(* IEC 61131-3 sources: LStream-JSON-XML/src/LStream (part 2) *)

(* ---- LStream_XmlDeserializer.st ---- *)
//region BLOCK INFO HEADER
    //===============================================================================
    // SIEMENS AG / (c)Copyright 2024
    //-------------------------------------------------------------------------------
    // Title:            LStream_XmlDeserializer
    // Comment/Function: parses a XML string provided in the Raw parameter
    //                   and rebuilds the contained tree structure
    // Library/Family:   LStream
    // Author:           DI FA S SUP E&C
    // Tested with:      S7-1500 V3.1
    // Engineering:      Simatic AX
    // Restrictions:     --
    // Requirements:     LStream_FindStringInByteArrayAdv(FC), LStream_typeElement(UDT)
    //-------------------------------------------------------------------------------
    // Change log table:
    // Version  | Date       | Expert in charge | Changes applied
    //----------|------------|------------------|------------------------------------
    // 01.00.00 | 2021-03-10 | DI FA S SUP E&C  | First released version
    // 01.06.00 | 2023-04-10 | DI FA S SUP E&C  | Rework and refactoring of entire library
    // 02.00.00 | 2024-11-11 | DI FA S SUP E&C  | Migrate library to Simatic AX
    //===============================================================================

//end_region
USING System.Timer;
USING System.Strings;
USING Simatic.Ax.LStream.Utilities;
USING Simatic.Ax.LStream.Models;
NAMESPACE Simatic.Ax.LStream
    FUNCTION_BLOCK LStream_XmlDeserializer
        VAR_INPUT
            /// Rising edge starts action once
            execute : BOOL;
            /// TRUE: Searches raw data for the value of the provided tree keys
            search  : BOOL;
        END_VAR
        VAR_OUTPUT
            /// TRUE: Commanded functionality has been completed successfully
            done : BOOL;
            /// TRUE: FB is not finished and new output values can be expected
            busy : BOOL;
            /// TRUE: An error occurred during the execution of the FB
            error : BOOL;
            /// 16#0000 - 16#7FFF: Status of the FB, 16#8000 - 16#FFFF: Error identification
            status : WORD := STATUS_NO_CALL;
            /// Current parse position in the raw XML data
            pointer : DINT;
            /// Count of parsed XML elements
            resultCount : DINT;
        END_VAR
        VAR_IN_OUT
            /// Tree parsed information is written to, if search option active, keys must be provided
            tree : ARRAY [*] of LStream_typeElement;
            /// Byte array of raw xml data
            raw : ARRAY[*] of BYTE;
        END_VAR
        VAR PUBLIC
            TimeoutTimer : System.Timer.OnDelay;
        END_VAR
        VAR
            /// Old value of 'execute' input for edge detection
            statOldExecute : BOOL;
            /// Static value of xml depth
            statDepth : SINT := SINT#-1;
            /// Static value of error
            statError : BOOL;
            /// Static value of busy
            statBusy : BOOL;
            /// Static value of status
            statStatus : WORD := STATUS_NO_CALL;
            /// Static value of fb state
            statFBState : USINT := FB_STATE_NO_PROCESSING;
            /// Static value of done
            statDone : BOOL;
            /// Static value of result count
            statResultCount : UINT;
            /// Static value of raw index
            statRawIndex : INT;
            /// Static value of tree index
            statTreeIndex : UINT;
            /// Static count of tree fields
            statCountOfTree : INT;
            /// Static count of raw fields
            statCountOfRaw : INT;
            /// TRUE: key is open, internal flag
            statIsKeyOpen : BOOL;
            /// TRUE: value is open, internal flag
            statIsValueOpen : BOOL;
            /// Determines the amount of open elements; if larger than 0 then at least one element is still open at the current parse position
            statElementOpen : UINT;
            /// TRUE: element is open, internal flag
            statIsElementOpen : BOOL;
            /// Current  information length key or value
            statInfoLen : UINT;
            /// Start index of current info in raw key or value
            statInfoStartIndex : INT;
            /// TRUE: Current key has already been written to the tree
            statKeyWritten: BOOL;
            /// Static key string
            statKey : STRING;
            /// Static value string
            statValue : STRING;
            /// TRUE: Only keys provided in tree will be parsed
            statSearch : BOOL;
            /// TRUE: Key exists in raw data
            statKeyFound : BOOL;
            /// Count of provided keys that weren't found
            statKeyNotFoundCount : UINT;
            /// Static search index
            statSearchIndex : DINT;
            /// Backtrack array for getting the last elements open
            statOpenElements : ARRAY[0.. MAX_CONCURRENT_OPEN_ELEMENTS] of UINT;
            /// Delimiter for attributes
            statAttrDelimiter : BYTE := BYTE#00;
        END_VAR
        VAR_TEMP
            /// Index of raw field
            tempRawIndex : INT;
            /// Temp of input execute
            tempExecute : BOOL;
            /// Provided key to which the value should be found
            tempKeyToFind : STRING;
            /// Temp value of search result
            tempSearchResult : DINT;
            /// Temp value of a byte for searching / looping
            tempChar : BYTE;
        END_VAR
        VAR CONSTANT
            /// FB state no processing, ideal state
            FB_STATE_NO_PROCESSING : USINT := USINT#0;
            /// FB state parse xml
            FB_STATE_PARSE : USINT := USINT#10;
            /// NO error - execution finished without errors
            STATUS_EXECUTION_FINISHED : WORD := WORD#16#0000;
            /// No job being currently processed
            STATUS_NO_CALL : WORD := WORD#16#7000;
            /// First call after incoming new job (rising edge 'execute')
            STATUS_FIRST_CALL : WORD := WORD#16#7001;
            /// Subsequent call during active processing without further details
            STATUS_SUBSEQUENT_CALL : WORD := WORD#16#7002;
            /// Error: provided array to too small
            ERR_TREE_ARRAY_TOO_SMALL : WORD := WORD#16#8201;
            /// Error: no raw data provided
            ERR_EMPTY_RAW_DATA : WORD := WORD#16#8401;
            /// Error: Encountered more closing tags than there are opening tags
            ERR_UNMATCHED_ELEMENT_CLOSE : WORD := WORD#16#8402;
            /// Error: Encountered an unexpected quotes character
            ERR_UNEXPECTED_QUOTES : WORD := WORD#16#8404;
            /// Error: Collection of all not further specified errors, e.g. unclosed elements before file end etc.
            ERR_MALFORMED : WORD := WORD#16#8406;
            /// Error: due to an undefined state in state machine
            ERR_UNDEFINED_STATE : WORD := WORD#16#8600;
            /// ASCII code for Unit Separator which is numerically the highest control character
            CONTROL_CHARACTERS_UPPER : WORD := WORD#16#1F;
            /// ASCII code for ? indicates xml header
            QUESTIONMARK : BYTE := BYTE#16#3F;
            /// ASCII code for ! indicates comment
            EXCLAMATION : BYTE := BYTE#16#21;
            /// ASCII code for " frames value
            DOUBLE_QUOTES : BYTE := BYTE#16#22;
            /// ASCII code for ' frames value
            QUOTES : BYTE := BYTE#16#27;
            /// ASCII code for < indicates a new key
            SMALLER : BYTE := BYTE#16#3C;
            /// ASCII code for '=' indicates key is finished follows by value
            EQUALS : BYTE := BYTE#16#3D;
            /// ASCII code for  > indicates key can be written
            GREATER : BYTE := BYTE#16#3E;
            /// ASCII code for SPACE indicates key is finished
            SPACE : BYTE := BYTE#16#20;
            /// ASCII code for / indicates closing
            SLASH : BYTE := BYTE#16#2F;
            /// ASCII code for carriage return
            CARRIAGE_RETURN : BYTE := BYTE#16#0D;
            /// ASCII code for line feed
            LINE_FEED : BYTE := BYTE#16#0A;
            /// ASCII code for TAB
            TAB : BYTE := BYTE#16#09;
            /// ASCII code for -
            MINUS : BYTE := BYTE#16#2D;
            /// Constant for zero value
            EMPTY : SINT := SINT#0;
            /// Numerical identifier for XML type element
            ELEMENT : SINT := SINT#0;
            /// Numerical identifier for XML type attribute
            ATTRIBUTE : SINT := SINT#1;
            /// Constant for first array dimension
            FIRST_DIM : USINT := USINT#1;
            /// Max duration of loop, will be continued in next cycle
            MAX_LOOP_TIME : TIME := T#3ms;
            /// Return value if Search in LStream_FindStringInByteCharArrayAdv was not successful
            INVALID_SEARCH : DINT := -1;
            /// String value in case key wasn't found
            KEY_NOT_FOUND : STRING := 'Key not found';
            /// String is default empty with string content named 'NULL'
            STRING_NULL : STRING := 'NULL';
            /// Maximal number of elements that can be open at any time
            MAX_CONCURRENT_OPEN_ELEMENTS : UINT := UINT#150;
            /// Empty string for resetting of fields
            STRING_EMPTY : STRING := '';

            /// ASCII code for ?
            QUESTIONMARK_INT : INT := 63;
            /// ASCII code for !
            EXCLAMATION_INT : INT := 33;
            /// ASCII code for "
            DOUBLE_QUOTES_INT : INT := 34;
            /// ASCII code for '
            QUOTES_INT : INT := 39;
            /// ASCII code for <
            SMALLER_INT : INT := 60;
            /// ASCII code for =
            EQUALS_INT : INT := 61;
            /// ASCII code for >
            GREATER_INT : INT := 62;
            /// ASCII code for SPACE
            SPACE_INT : INT := 32;
            /// ASCII code for /
            SLASH_INT : INT := 47;
            /// ASCII code for carriage return
            CARRIAGE_RETURN_INT : INT := 13;
            /// ASCII code for line feed
            LINE_FEED_INT : INT := 10;
            /// ASCII code for TAB
            TAB_INT : INT := 9;
            /// ASCII code for -
            MINUS_INT : INT := 45;
        END_VAR
        tempExecute := execute;

    //region TRIGGERING

        IF ((tempExecute = TRUE) AND (statOldExecute = FALSE) AND (statStatus = STATUS_NO_CALL)) THEN

            //First call; Initialize FB
            statDone := FALSE;
            statBusy := TRUE;
            statStatus := STATUS_FIRST_CALL;

            //Initialize functionality: reset of variables, diagnostics, etc.
            statSearch := search;
            statCountOfRaw := TO_INT(UPPER_BOUND(raw, FIRST_DIM));
            statCountOfTree := TO_INT(UPPER_BOUND(tree, FIRST_DIM));
            statTreeIndex := TO_UINT(LOWER_BOUND(tree, FIRST_DIM));
            statDepth := SINT#0;
            statRawIndex := 0;
            statIsKeyOpen := FALSE;
            statIsValueOpen := FALSE;
            statIsElementOpen := FALSE;
            statElementOpen := UINT#0;
            statKeyWritten := FALSE;
            statInfoLen := UINT#0;
            statInfoStartIndex := 0;
            statKey := '';
            statValue := '';
            statKeyFound := FALSE;
            statSearchIndex := 0;
            statKeyNotFoundCount := UINT#0;

            // State machine - start processing
            statFBState := FB_STATE_PARSE;

            IF (NOT (statCountOfRaw > EMPTY)) THEN
                statStatus := ERR_EMPTY_RAW_DATA;
            END_IF;

            FOR tempRawIndex := TO_INT(statTreeIndex) TO statCountOfTree DO

                tree[tempRawIndex].types := SINT#-1;
                tree[tempRawIndex].depth := SINT#-1;
                tree[tempRawIndex].key := STRING_EMPTY;
                tree[tempRawIndex].value := STRING_NULL;

            END_FOR;
        ELSIF (statStatus = STATUS_FIRST_CALL) THEN
            statStatus := STATUS_SUBSEQUENT_CALL;
        END_IF;

        // Edge detection 'execute' input
        statOldExecute := tempExecute;

    //endRegion TRIGGERING
        IF (statStatus = STATUS_NO_CALL) THEN // Nothing to do -> End here to reduce "system load"
            RETURN;
        END_IF;
    //region PROGRAM LOGIC

        CASE statFBState OF
            FB_STATE_NO_PROCESSING:
                // #region NO PROCESSING
                    // No processing active (Note: this state must always be present AND left empty)
                    ;
                // #endregion NO PROCESSING
            FB_STATE_PARSE:
                // #region PARSE XML

                    //reset and start watchdog here so that for loop runs for a maximum of 5 seconds
                    TimeoutTimer(signal := FALSE, duration := MAX_LOOP_TIME);

                    //start watchdog
                    TimeoutTimer(signal := TRUE, duration := MAX_LOOP_TIME);

                    tempRawIndex := statRawIndex;

                    WHILE tempRawIndex <= statCountOfRaw DO
                        //pre check if key exist in raw data, only if search option is active and key wasn't already found
                        IF (statSearch AND statKeyFound = FALSE) THEN
                            IF (TO_DINT(statTreeIndex) < statCountOfTree) THEN              //Convert to DINT to prevent possible overflows
                                tempSearchResult := LStream_FindStringInByteCharArrayAdv(searchFor := tree[statTreeIndex].key, startPosition := statSearchIndex, searchIn := raw);

                                IF tempSearchResult = INVALID_SEARCH THEN
                                    // Case key not found
                                    tree[statTreeIndex].value := KEY_NOT_FOUND;
                                    statTreeIndex := statTreeIndex + UINT#1;
                                    statKeyNotFoundCount := statKeyNotFoundCount + UINT#1;
                                ELSE
                                    // Case key found
                                    // move read pointer to last found index
                                    statSearchIndex := tempSearchResult;
                                    statKeyFound := TRUE;
                                END_IF;
                            END_IF;
                        END_IF;

                        statRawIndex := tempRawIndex;
                        // Switch case of current byte
                        CASE TO_INT(raw[tempRawIndex]) OF           //BYTE/ WORD Can not be selected as CASE selector
                            SMALLER_INT:
                                //region READ OPENING KEY SYMBOLS

                                    // There MUST be some characters after an open <
                                    // so if the array is too short the xml is malformed
                                    IF ((tempRawIndex + 1) > statCountOfRaw) THEN
                                        statStatus := ERR_MALFORMED;
                                        statDone := TRUE;
                                        EXIT;
                                    END_IF;
                                    IF statIsValueOpen
                                        AND statInfoLen > UINT#0
                                        AND tree[statOpenElements[statElementOpen]].value = STRING_NULL
                                        AND raw[statInfoStartIndex] <> SMALLER
                                    THEN
                                        //region WRITE VALUE
                                        IF statInfoLen < UINT#0 THEN
                                            statValue := STRING_EMPTY;
                                        ELSE
                                            CharsToString(chars := raw,
                                                        startPosition := statInfoStartIndex,
                                                        length:= statInfoLen,
                                                        result => statValue);
                                        END_IF;

                                        tree[statOpenElements[statElementOpen]].value := statValue;

                                        statInfoLen := UINT#0;
                                        statIsValueOpen := FALSE;

                                        //endregion WRITE VALUE
                                    END_IF;

                                    // Check if is XML Header or comment by looking ahead by one
                                    IF (raw[tempRawIndex +1] = QUESTIONMARK) OR (raw[tempRawIndex + 1] = EXCLAMATION) THEN

                                        CASE TO_INT(raw[tempRawIndex + 1]) OF                   //SAME CASE BYTE NOT ALLOWED
                                            EXCLAMATION_INT:
                                                IF raw[tempRawIndex +2] = MINUS THEN
                                                    tempChar := MINUS;
                                                ELSE
                                                    tempChar := GREATER;
                                                END_IF;
                                            QUESTIONMARK_INT:
                                                tempChar := QUESTIONMARK;
                                        END_CASE;

                                        //region IS IGNORABLE

                                            // At least two more characters have to be in the XML otherwise it is malformed
                                            // <? ?>

                                            IF tempRawIndex + 2 > statCountOfRaw THEN
                                                statStatus := ERR_MALFORMED;
                                                statDone := TRUE;
                                                EXIT;
                                            END_IF;
                                            IF tempRawIndex + 2 <= statCountOfRaw THEN
                                                tempRawIndex := tempRawIndex + 2;

                                                // Iterate until either ? or ! are found or until the end of the raw array is
                                                // reached; if the end of the array has been reached before the end of the
                                                // header or comment then the XML must be malformed and therefore a error
                                                // is set in the status
                                                WHILE raw[tempRawIndex] <> tempChar AND raw[tempRawIndex] <> GREATER DO
                                                    IF tempRawIndex + 1 > statCountOfRaw THEN
                                                        statStatus := ERR_MALFORMED;
                                                        statDone := TRUE;
                                                        EXIT;
                                                    END_IF;

                                                    IF raw[tempRawIndex + 1] = GREATER THEN
                                                        EXIT;
                                                    END_IF;

                                                    tempRawIndex := tempRawIndex + 1;

                                                END_WHILE;

                                                // End of a comment, meaning that there has to be at least one more MINUS
                                                // before comment can be closed
                                                IF tempChar = MINUS THEN

                                                    IF tempRawIndex + 1 > statCountOfRaw THEN
                                                        statStatus := ERR_MALFORMED;
                                                        statDone := TRUE;
                                                        EXIT;
                                                    END_IF;

                                                    tempRawIndex := tempRawIndex +1;
                                                END_IF;

                                                // Array ended before the comment or header could be closed which is illegal
                                                // In case the loop ran successfully we are here, which requires at least
                                                // one more character
                                                // <!-- Some Comment -->
                                                //                    ^
                                                //                    |
                                                //                    Current index

                                                IF statStatus.%X15 OR tempRawIndex + 1 > statCountOfRaw THEN
                                                    statStatus := ERR_MALFORMED;
                                                    statDone := TRUE;
                                                    EXIT;
                                                END_IF;

                                                IF raw[tempRawIndex + 1] <> GREATER THEN
                                                    statRawIndex := tempRawIndex;
                                                    statStatus := ERR_MALFORMED;
                                                    statDone := TRUE;
                                                    EXIT;
                                                END_IF;

                                                tempRawIndex := tempRawIndex +1;

                                            END_IF;

                                            statInfoLen := UINT#0;
                                            //rest length buffer
                                        //endregion IS IGNORABLE

                                        // Look ahead for closing otherwise open element
                                    ELSIF (raw[tempRawIndex + 1] <> SLASH) THEN

                                        // Indicates opening of element
                                        //region OPENING OF ELEMENT
                                            IF (TO_DINT(statTreeIndex) > statCountOfTree + 1) THEN              //CONVERSION TO DINT
                                                // data does not fit in the provided tree
                                                statStatus := ERR_TREE_ARRAY_TOO_SMALL;
                                                statDone := TRUE;
                                                EXIT;
                                            END_IF;

                                            IF statElementOpen + UINT#1 > MAX_CONCURRENT_OPEN_ELEMENTS THEN
                                                statStatus := ERR_MALFORMED;
                                                statDone := TRUE;
                                                pointer := tempRawIndex;
                                                EXIT;
                                            END_IF;

                                            // new element
                                            statElementOpen := statElementOpen + UINT#1; // increment the opened element count as a new element is "created" here

                                            statOpenElements[statElementOpen] := statTreeIndex;
                                            statIsValueOpen := FALSE;
                                            statDepth := statDepth + SINT#1;
                                            statInfoStartIndex := tempRawIndex + 1;
                                            statInfoLen := UINT#0;

                                            // Invalid as the xml can not stop after opening
                                            // <a>v</a><EOF
                                            //         ^
                                            //         | current

                                            IF tempRawIndex + 1 > statCountOfRaw THEN
                                                statStatus := ERR_MALFORMED;
                                                statDone := TRUE;
                                                pointer := tempRawIndex;
                                                EXIT;
                                            END_IF;

                                            tempRawIndex := tempRawIndex +1;

                                            //Region READ KEY OF NEW ELEMENT
                                                WHILE raw[tempRawIndex] <> SPACE AND raw[tempRawIndex] <> LINE_FEED
                                                    AND raw[tempRawIndex] <> CARRIAGE_RETURN
                                                    AND raw[tempRawIndex] <> TAB
                                                    AND raw[tempRawIndex] <> SMALLER
                                                    AND raw[tempRawIndex] <> BYTE#16#00
                                                    AND raw[tempRawIndex] <> GREATER
                                                    AND raw[tempRawIndex] > CONTROL_CHARACTERS_UPPER
                                                    AND raw[tempRawIndex] <> SLASH
                                                DO
                                                    IF tempRawIndex + 1 > statCountOfRaw THEN
                                                        statStatus := ERR_MALFORMED;
                                                        statDone := TRUE;
                                                        pointer := tempRawIndex;
                                                        EXIT;
                                                    END_IF;

                                                    statInfoLen := statInfoLen + UINT#1;
                                                    tempRawIndex := tempRawIndex + 1;
                                                END_WHILE;

                                                IF statStatus.%X15 OR statInfoLen = UINT#0 THEN
                                                    statStatus := ERR_MALFORMED;
                                                    statDone := TRUE;
                                                    pointer := tempRawIndex;
                                                    EXIT;
                                                END_IF;

                                                IF (TO_DINT(statTreeIndex) > statCountOfTree) THEN
                                                    //data does not fit in the provided tree
                                                    statStatus := ERR_TREE_ARRAY_TOO_SMALL;
                                                    statDone := TRUE;
                                                    EXIT;
                                                END_IF;

                                                CharsToString(chars := raw,
                                                            startPosition := statInfoStartIndex,
                                                            length := statInfoLen,
                                                            result => statKey);
                                                IF (statSearch) THEN
                                                    //only write into tree, if key matches, otherwise continue with search for matching key
                                                    IF (statKey = tree[statTreeIndex].key) THEN
                                                        tree[statTreeIndex].depth := statDepth;
                                                        tree[statTreeIndex].types := ELEMENT;
                                                        statTreeIndex := statTreeIndex + UINT#1;
                                                        statKeyFound := FALSE;
                                                    END_IF;

                                                ELSE  // if search option isn't active (parse all) the add key to the current tree index
                                                    tree[statTreeIndex].key := statKey;
                                                    tree[statTreeIndex].types := ELEMENT;
                                                    tree[statTreeIndex].depth := statDepth;
                                                    statTreeIndex := statTreeIndex + UINT#1;
                                                    statKeyFound := FALSE;
                                                    statKeyWritten := TRUE;
                                                    statIsKeyOpen := FALSE;
                                                END_IF;
                                            //endregion READ KEY OF NEW ELEMENT

                                            statKeyWritten := FALSE;

                                            IF raw[tempRawIndex] = SLASH THEN
                                                statOpenElements[statElementOpen] := UINT#0;
                                                statElementOpen := statElementOpen - UINT#1;

                                                statIsValueOpen := FALSE;
                                                statDepth := statDepth - SINT#1;

                                                tempRawIndex := tempRawIndex +  1;

                                            ELSIF raw[tempRawIndex] = GREATER THEN
                                                statIsValueOpen := TRUE;
                                            ELSE
                                                statIsKeyOpen := TRUE;
                                            END_IF;

                                            statInfoStartIndex := tempRawIndex + 1;
                                            statInfoLen := UINT#0;
                                        //endregion OPENING OF ELEMENT
                                    ELSE
                                        statIsValueOpen := FALSE;
                                    END_IF;

                                //endregion READ OPENING KEY SYMBOLS

                            SLASH_INT:
                                //region READ DELIMITER /
                                    IF statIsValueOpen THEN

                                        statInfoLen := statInfoLen + UINT#1;

                                    ELSE

                                        IF statElementOpen <= UINT#0 THEN

                                            statStatus := ERR_UNMATCHED_ELEMENT_CLOSE;
                                            statDone := TRUE;
                                            EXIT;

                                        END_IF;

                                        statDepth := statDepth - SINT#1;
                                        statInfoLen := UINT#0;
                                        IF statElementOpen >= UINT#0 THEN
                                            statOpenElements[statElementOpen] := UINT#0;
                                        END_IF;

                                        statElementOpen := statElementOpen - UINT#1;
                                        // Skip everything in the element key until the end of the key
                                        //
                                        // </elementkey>
                                        //  ^          ^
                                        //  |          |
                                        //  current    skip position
                                        WHILE raw[tempRawIndex] <> GREATER DO

                                            IF tempRawIndex + 1 > statCountOfRaw THEN
                                                statStatus := ERR_MALFORMED;
                                                statDone := TRUE;
                                                EXIT;
                                            END_IF;

                                            tempRawIndex := tempRawIndex + 1;

                                        END_WHILE;

                                        // So that next iteration will be on the greater than > sign
                                        // </element>
                                        //         ^
                                        //         |
                                        //         Current index
                                        tempRawIndex := tempRawIndex - 1;

                                        // Array ended unexpected and is therefore malformed
                                        IF statStatus.%X15 THEN
                                            statStatus := ERR_MALFORMED;
                                            statDone := TRUE;
                                            EXIT;
                                        END_IF;

                                    END_IF;
                            //endregion READ DELIMITER /

                        SPACE_INT:

                            IF statIsValueOpen THEN

                                statInfoLen := statInfoLen + UINT#1;

                            ELSIF statIsKeyOpen THEN

                                tempRawIndex := tempRawIndex; // Ignore "empty space" between a key name and '=' so spaces are not added to the key

                            ELSE
                                statIsKeyOpen := TRUE;
                                statInfoStartIndex := tempRawIndex + 1;
                                statInfoLen := UINT#0;
                            END_IF;

                        GREATER_INT:
                            //region READ WRITING KEY SYMBOLS

                                IF NOT statIsValueOpen THEN
                                    statIsValueOpen := TRUE;
                                    statInfoStartIndex := tempRawIndex + 1;
                                    statInfoLen := UINT#0;
                                ELSE
                                    statInfoLen := statInfoLen + UINT#1;
                                END_IF;

                            //endregion READ WRITING KEY SYMBOLS

                        EQUALS_INT:

                            IF statIsValueOpen THEN

                                statInfoLen := statInfoLen + UINT#1;

                            ELSIF statIsKeyOpen THEN

                                IF (TO_DINT(statTreeIndex) > statCountOfTree) THEN
                                    //data does not fit in the provided tree
                                    statStatus := ERR_TREE_ARRAY_TOO_SMALL;
                                    statDone := TRUE;
                                    EXIT;
                                END_IF;

                                CharsToString(chars := raw,
                                            startPosition := statInfoStartIndex,
                                            length := statInfoLen,
                                            result => statKey);

                                IF (statSearch) THEN
                                    //only write into tree, if key matches, otherwise continue with search for matching key
                                    IF (statKey = tree[statTreeIndex].key) THEN
                                        tree[statTreeIndex].depth := statDepth;
                                        tree[statTreeIndex].types := ATTRIBUTE;
                                        statTreeIndex := statTreeIndex + UINT#1;
                                        statKeyFound := FALSE;
                                    END_IF;

                                ELSE// if search option isn't active (parse all) the add key to the current tree index
                                    tree[statTreeIndex].key := statKey;
                                    tree[statTreeIndex].types := ATTRIBUTE;
                                    tree[statTreeIndex].depth := statDepth;
                                    statTreeIndex := statTreeIndex + UINT#1;
                                    statKeyFound := FALSE;
                                    statKeyWritten := TRUE;

                                END_IF;

                                statIsKeyOpen := FALSE;
                                statInfoStartIndex := tempRawIndex + 1;
                                statInfoLen := UINT#0;

                            END_IF;

                            IF NOT statIsValueOpen THEN

                                IF tempRawIndex + 1 > statCountOfRaw THEN
                                    statStatus := ERR_MALFORMED;
                                    statDone := TRUE;
                                    pointer := tempRawIndex;
                                    EXIT;
                                END_IF;

                                tempRawIndex := tempRawIndex + 1;

                                WHILE raw[tempRawIndex] = SPACE
                                    OR raw[tempRawIndex] = LINE_FEED
                                    OR raw[tempRawIndex] = CARRIAGE_RETURN
                                    OR raw[tempRawIndex] = TAB
                                DO

                                    IF tempRawIndex + 1 > statCountOfRaw THEN
                                        statStatus := ERR_MALFORMED;
                                        statDone := TRUE;
                                        pointer := tempRawIndex;
                                        EXIT;
                                    END_IF;

                                    tempRawIndex := tempRawIndex + 1;

                                END_WHILE;

                                // This is not valid, as a equals character '=' that is not within an element
                                // has to open an attribute with either ' or "
                                IF raw[tempRawIndex] <> DOUBLE_QUOTES AND raw[tempRawIndex] <> QUOTES THEN

                                    statStatus := ERR_MALFORMED;
                                    statDone := TRUE;
                                    pointer := tempRawIndex;
                                    EXIT;

                                END_IF;

                                statAttrDelimiter := raw[tempRawIndex];

                                IF tempRawIndex + 1 > statCountOfRaw THEN
                                    statStatus := ERR_MALFORMED;
                                    statDone := TRUE;
                                    pointer := tempRawIndex;
                                    EXIT;
                                END_IF;

                                tempRawIndex := tempRawIndex + 1;

                                statInfoLen := UINT#0;
                                statInfoStartIndex := tempRawIndex;

                                WHILE raw[tempRawIndex] <> statAttrDelimiter DO

                                    IF tempRawIndex + 1 > statCountOfRaw OR raw[tempRawIndex] = SMALLER THEN
                                        statStatus := ERR_MALFORMED;
                                        statDone := TRUE;
                                        pointer := tempRawIndex;
                                        EXIT;
                                    END_IF;

                                    tempRawIndex := tempRawIndex + 1;
                                    statInfoLen := statInfoLen + UINT#1;

                                END_WHILE;

                                IF statStatus.%X15 THEN
                                    EXIT;
                                END_IF;

                                IF statInfoLen <= UINT#0 THEN
                                    statValue := STRING_EMPTY;
                                ELSE
                                    //attach value to last key node
                                    CharsToString(chars := raw,
                                                startPosition := statInfoStartIndex,
                                                length := statInfoLen,
                                                result => statValue);
                                END_IF;

                                IF (statSearch) THEN
                                    //only write into tree, if key matches, otherwise continue with search for matching key
                                    IF (statKey = tree[statTreeIndex - UINT#1].key) THEN
                                        tree[statTreeIndex - UINT#1].depth := statDepth;
                                        tree[statTreeIndex - UINT#1].value := statValue;
                                        tree[statTreeIndex - UINT#1].types := ATTRIBUTE;
                                    END_IF;
                                ELSE
                                    // if search option isn't active (parse all) the add key to the current tree index
                                    tree[statTreeIndex - UINT#1].value := statValue;
                                    tree[statTreeIndex - UINT#1].types := ATTRIBUTE;
                                    tree[statTreeIndex - UINT#1].depth := statDepth;

                                    statIsValueOpen := false;
                                END_IF;

                            END_IF;

                        QUOTES_INT:
                            //region READ VALUE SYMBOLS
                                // Quotes can never occur within a key, which is always closed by a '=', '/>' or '>'
                                IF statIsKeyOpen THEN
                                    statStatus := ERR_UNEXPECTED_QUOTES;
                                    statDone := TRUE;
                                    pointer := tempRawIndex;
                                    EXIT;
                                END_IF;

                                statInfoLen := statInfoLen + UINT#1;

                            //endregion READ VALUE SYMBOLS

                        ELSE//all other characters
                            //region READ OTHER SIGN

                                statInfoLen := statInfoLen + UINT#1;

                            //endregion READ OTHER SIGN
                        END_CASE;

                        statRawIndex := tempRawIndex;

                        // Call for Timeout timer to update value
                        TimeoutTimer();
                        //quit and resume in next cycle if watchdogtimer is exceed
                        IF (TimeoutTimer.output) THEN
                            statRawIndex := statRawIndex + 1;
                            EXIT;
                        ELSIF tempRawIndex <= statCountOfRaw THEN
                            tempRawIndex := tempRawIndex + 1;
                        END_IF;
                    END_WHILE;

                    //if parser is through the entire raw data or end of tree array reached
                    IF (statRawIndex >= statCountOfRaw) OR (TO_DINT(statTreeIndex) > statCountOfTree) THEN
                        statStatus := STATUS_EXECUTION_FINISHED;
                        statResultCount := statTreeIndex - statKeyNotFoundCount;
                    END_IF;

                //endregion PARSE XML

            ELSE // Undefined state in state machine reached
                //region UNDEFINED STATE
                    statStatus := ERR_UNDEFINED_STATE;
                //endregion UNDEFINED STATE
        END_CASE;

    //endregion PROGRAM LOGIC

    //region OUTPUTS

        //Write Outputs
        IF (statStatus = STATUS_EXECUTION_FINISHED) AND (statDone = FALSE) THEN // Execution finished without errors
            //region EXECUTION FINISHED
                statDone := TRUE;
                statBusy := FALSE;
                statError := FALSE;
                // execution aborted --> set state no processing
                statFBState := FB_STATE_NO_PROCESSING;
            //endregion EXECUTION FINISHED

        ELSIF (statStatus.%X15 = TRUE) AND (statError = FALSE) THEN // Error occurred (#statStatus is 16#8000 to 16#FFFF)
            //region ERROR OCCURRED
                statDone := FALSE;
                statBusy := FALSE;
                statError := TRUE;
                // execution aborted --> set state no processing
                statFBState := FB_STATE_NO_PROCESSING;
            //endregion ERROR OCCURRED

        ELSIF (tempExecute = FALSE) AND ((statDone = TRUE) OR (statError = TRUE)) THEN // Reset outputs
            //region EXECUTE RESET
                statDone := FALSE;
                statBusy := FALSE;
                statError := FALSE;
                statStatus := STATUS_NO_CALL;
                // Reset application specific outputs
                statResultCount := UINT#0;
            //endregion EXECUTE RESET
        END_IF;

        //region WRITE STATIC VALUES TO OUTPUTS
            // write application specific temp values to outputs
            resultCount := TO_INT(statResultCount);
            done := statDone;
            error := statStatus.%X15;
            status := statStatus;
            busy := statBusy;
        //endregion WRITE STATIC VALUES TO OUTPUTS

    //endregion OUTPUTS
    END_FUNCTION_BLOCK

END_NAMESPACE

(* ---- LStream_XmlSerializer.st ---- *)
//region BLOCK INFO HEADER
    //===============================================================================
    // SIEMENS AG / (c)Copyright 2024
    //-------------------------------------------------------------------------------
    // Title:            LStream_XmlSerializer
    // Comment/Function: FB converts prefilled array of udt LParse_typeElement to a xml structure.
    //                   XML structure is returned as a Byte array
    // Library/Family:   LStream
    // Author:           DI FA S SUP E&C
    // Tested with:      S7-1500 V3.1
    // Engineering:      Simatic AX
    // Restrictions:     --
    // Requirements:     LStream_WriteOutString(FC), LStream_typeElement(UDT)
    //-------------------------------------------------------------------------------
    // Change log table:
    // Version  | Date       | Expert in charge | Changes applied
    //----------|------------|------------------|------------------------------------
    // 01.00.00 | 2021-03-10 | DI FA S SUP E&C  | First released version
    // 01.06.00 | 2023-04-10 | DI FA S SUP E&C  | Rework and refactoring of entire library
    // 02.00.00 | 2024-11-11 | DI FA S SUP E&C  | Migrate library to Simatic AX
    //===============================================================================

//end_region
USING System.Timer;
USING Simatic.Ax.LStream.Utilities;
USING System.Strings;
USING Simatic.Ax.LStream.Models;
NAMESPACE Simatic.Ax.LStream
    FUNCTION_BLOCK LStream_XmlSerializer
        VAR_INPUT
            /// Rising edge starts action once
            execute : BOOL;
        END_VAR
        VAR_OUTPUT
            /// TRUE: Commanded functionality has been completed successfully
            done : BOOL;
            /// TRUE: FB is not finished and new output values can be expected
            busy : BOOL;
            /// TRUE: An error occurred during the execution of the FB
            error : BOOL;
            /// 16#0000 - 16#7FFF: Status of the FB, 16#8000 - 16#FFFF: Error identification
            status : WORD := STATUS_NO_CALL;
            /// Count of char/ byte info elements in byte array
            count : UINT;
        END_VAR
        VAR_IN_OUT
            /// Describes the element for LStream libraries, by providing key-value pair and the depth of the element
            tree : ARRAY [*] of LStream_typeElement;
            /// XML structure as array of bytes
            xmlByteArray : ARRAY[*] of BYTE;
        END_VAR
        VAR PUBLIC
            TimeoutTimer : System.Timer.OnDelay;
        END_VAR
        VAR
            /// Old value of 'execute' input for edge detection
            statExecuteOld : BOOL;
            /// Static value for output 'done'
            statDone : BOOL;
            /// Static value for output 'busy'
            statBusy : BOOL;
            /// Static value for output 'error'
            statError : BOOL;
            /// Static value for output 'count'
            statCount : UINT;
            /// Static value for output 'status'
            statStatus : WORD := STATUS_NO_CALL;
            /// State in the state machine of the FB
            statFBState : DINT := FB_STATE_NO_PROCESSING;
            /// Previous state in the state machine of the FB
            statFBPreviousState : DINT := FB_STATE_NO_PROCESSING;
            /// Next state in the state machine of the FB
            statFBNextState : DINT := FB_STATE_NO_PROCESSING;
            /// Index indicating current element of byte array to be written
            statIndexXmlByteArray : UINT;
            /// Index indicating current element of tree array to be read
            statIndexTreeArray : UINT;
            /// Length of tree array
            statTreeLen : DINT;
            /// Length of xml byte array
            statXmlByteLen : DINT;
            /// Static value of current information that should be written to XML
            statInfoToWrite : STRING;
            /// TRUE: is last element in tree array
            statIsLastElement : BOOL;
            /// Stack of open elements
            statStackIndexOpenElement : ARRAY[0..STACK_SIZE] OF UINT;
            /// Stack pointer
            statStackIndex : INT := -1;
            /// Depth of the current tree element
            statCurrentDepth : INT;
            statWorkingDepth : INT;
        END_VAR
        VAR_TEMP
            /// Temporary value for input 'execute'
            tempExecute : BOOL;
            /// Temporary value indicating count of chars added to byte array
            tempCntCharsAdded : INT;
            /// Temporary iterator value
            tempIterator : UINT;
            /// Temporary value indicating that the current element has nested elements
            tempHasNested : BOOL;
        END_VAR
        VAR CONSTANT
            /// FB state: No processing
            FB_STATE_NO_PROCESSING : DINT := 0;
            /// FB state: Clean the entire byte array
            FB_STATE_CLEAR_BYTE_ARRAY : DINT := 1;
            /// FB state: Write XML Header
            FB_STATE_XML_HEADER : DINT := 2;
            /// FB state: Get Next Element
            FB_STATE_NEXT_ELEMENT : DINT := 3;
            /// FB state: Switch Element type
            FB_STATE_ELEMENT_TYPE_OPEN : DINT := 4;
            /// FB state: Add Information to xml byte array
            FB_STATE_WRITE_TO_XML : DINT := 5;
            /// FB state: Close Parent Element
            FB_STATE_CLOSE_STACK_ELEMENT : DINT := 6;
            /// FB state: Error
            FB_STATE_ERROR : DINT := 7;
            /// FB state: Done
            FB_STATE_DONE : DINT := 8;
            /// Execution finished without errors
            STATUS_EXECUTION_FINISHED : WORD := WORD#16#0000;
            /// No job being currently processed
            STATUS_NO_CALL : WORD := WORD#16#7000;
            /// First call after incoming new job (rising edge 'execute')
            STATUS_FIRST_CALL : WORD := WORD#16#7001;
            /// Subsequent call during active processing without further details
            STATUS_SUBSEQUENT_CALL : WORD := WORD#16#7002;
            /// Subsequent call during active processing without further details
            ERR_UNDEFINED_STATE : WORD := WORD#16#8600;
            /// Error: wrong operation of the function block
            ERR_IN_BLOCK_OPERATION : WORD := WORD#16#8601;
            /// Error: during parameterization
            ERR_PARAMETRIZATION : WORD := WORD#16#8200;
            /// Error: when processing from outside (e. g. wrong I/O signals, axis not referenced)
            ERR_PROCESSING_EXTERN : WORD := WORD#16#8400;
            /// Error: user enter undefined type
            ERR_UNDEFINED_TYPE : WORD := WORD#16#8401;
            /// Error: provided xml tree structure is too deep
            ERR_UNEXPECTED_DEPTH : WORD := WORD#16#8402;
            /// Error: provided xml tree structure does not contain correct depth
            ERR_DEPTH_MISSING : WORD := WORD#16#8403;
            /// Error: when processing internally (e. g. when calling a system function)
            ERR_PROCESSING_INTERN : WORD := WORD#16#8600;
            /// Error: tree array out of bounds
            ERR_TREE_OUT_OF_BOUNDS : WORD := WORD#16#8601;
            /// Error: byte array out of bounds
            ERR_XML_OUT_OF_BOUNDS : WORD := WORD#16#8602;
            /// Error: stack array out of bounds
            ERR_STACK_OUT_OF_BOUNDS : WORD := WORD#16#8603;
            /// Error: reserved area
            ERR_AREA_RESERVED : WORD := WORD#16#8800;
            /// Error: user-defined error classes
            ERR_USER_DEFINED_CLASSES : WORD := WORD#16#9000;
            /// Constant to increment by one
            INCREMENT_BY_ONE : SINT := SINT#1;
            /// Constant to decrement by one
            DECREMENT_BY_ONE : SINT := SINT#1;
            /// Numerical identifier for XML type element
            ELEMENT : SINT := SINT#0;
            /// Numerical identifier for XML type attribute
            ATTRIBUTE : SINT := SINT#1;
            /// Numerical identifier for XML type text
            TEXT : SINT := SINT#2;
            /// Constant for first array dimension
            FIRST_DIM : USINT := USINT#1;
            /// Max duration of loop, will be continued in next cycle
            MAX_REPEAT_TIME : TIME := T#6ms;
            /// XML Header, leads every XML File
            XML_HEADER : STRING := '<?xml version="1.0" encoding="ASCII"?>';
            /// ASCII code for < indicates a new key
            XML_KEY_OPEN : CHAR := '<';
            /// ASCII code for '=' indicates key is finished follows by value
            XML_ATTRIBUTE_OPEN : STRING := '="';
            /// ASCII code for  > indicates key can be written
            XML_KEY_CLOSE_GREATER : CHAR := '>';
            /// ASCII code for / indicates closing
            XML_KEY_CLOSE_SLASH : CHAR := '/';
            /// ASCII code  for " frames value
            XML_ATTRIBUTE_CLOSE : CHAR := '"';
            /// Constant value to get next index
            NEXT_INDEX : UINT := UINT#1;
            /// Constant for Stack Size, equals max depth
            STACK_SIZE : UINT := UINT#30;
            /// ASCII code for white space
            WHITE_SPACE: CHAR := ' ';
            /// Constant value representing not initialized tree element
            NOT_INITIALIZED : SINT := SINT#-1;
            /// String for NULL value
            NULL_CONST : STRING := STRING#'NULL';
            /// Empty string for checking if value is contained within the string
            EMPTY_STRING : STRING := STRING#'';
            /// Empty byte for cleaning the byte array
            EMPTY_BYTE : BYTE := BYTE#16#0;

        END_VAR;

        tempExecute := execute; // Work with temporary value / create process image

        //region TRIGGERING
            IF (tempExecute = TRUE) AND (statExecuteOld = FALSE) // Check if FB is triggered
                AND (statStatus = STATUS_NO_CALL)
            THEN // First call; initialize FB
                statDone := FALSE;
                statBusy := TRUE;
                statError := FALSE;
                statStatus := STATUS_FIRST_CALL;
                // State machine - start processing
                statFbState := FB_STATE_CLEAR_BYTE_ARRAY;

                //Initialize functionality: reset OF variables, diagnostics, etc.
                statXmlByteLen := UPPER_BOUND(xmlByteArray, FIRST_DIM);
                statTreeLen := UPPER_BOUND(tree, FIRST_DIM);
                statIndexTreeArray := UINT#0;
                statIndexXmlByteArray := UINT#0;
                statIsLastElement := FALSE;
                statStackIndex := -1;

                statCurrentDepth := tree[statIndexTreeArray].depth;

            ELSIF (statStatus = STATUS_FIRST_CALL) THEN
                statStatus := STATUS_SUBSEQUENT_CALL;
            END_IF;

            // Edge detection 'execute' input
            statExecuteOld := tempExecute;
        //endregion TRIGGERING

        IF (statStatus = STATUS_NO_CALL) THEN // Nothing to do -> End here to reduce "system load"
            RETURN;
        END_IF;

        //region STATE_MACHINE
            //rest and start watchdog here so that repeat until has a maximum duration of constant MAX_LOOP_TIME
            TimeoutTimer(signal := FALSE, duration := MAX_REPEAT_TIME);
            //start watchdog
            TimeoutTimer(signal := TRUE, duration := MAX_REPEAT_TIME);
            REPEAT
                statFbPreviousState := statFbState;

                CASE statFbState OF // State machine of FB

                    FB_STATE_NO_PROCESSING:
                        //region NO PROCESSING
                            // No processing active (Note: this state must always be present and left empty)
                            EXIT;
                        //endregion NO PROCESSING

                    FB_STATE_CLEAR_BYTE_ARRAY:
                        //region CLEAR BYTE ARRAY
                            WHILE TRUE DO

                                IF statIndexXmlByteArray > statXmlByteLen THEN
                                    EXIT;
                                END_IF;
                                xmlByteArray[statIndexXmlByteArray] := EMPTY_BYTE;
                                statIndexXmlByteArray := statIndexXmlByteArray + UINT#1;
                            END_WHILE;

                            statIndexXmlByteArray := tempIterator;
                            statFbState := FB_STATE_XML_HEADER;
                        //endregion CLEAR BYTE ARRAY
                    FB_STATE_XML_HEADER: // Add xml Header
                        //region WRITE XML HEADER
                            // Write XML Header at the beginning of byte array
                            statInfoToWrite := XML_HEADER;

                            //Move to state Write
                            tempCntCharsAdded := LStream_WriteOutString(offset := statIndexXmlByteArray, toWrite := statInfoToWrite, xmlByteArray := xmlByteArray);

                            IF tempCntCharsAdded = -1 THEN
                                statStatus := ERR_XML_OUT_OF_BOUNDS;
                                statFbState := FB_STATE_ERROR;
                                CONTINUE;
                            END_IF;

                            statIndexXmlByteArray := statIndexXmlByteArray + TO_UINT(tempCntCharsAdded) + UINT#1;

                            //Set state, that should be executed after writing
                            statFbState := FB_STATE_NEXT_ELEMENT;

                        //endregion WRITE XML HEADER

                    FB_STATE_NEXT_ELEMENT: // Get Next Element and write tree key
                        //region GET NEXT ELEMENT

                            IF statIndexTreeArray = UINT#204 THEN
                                statIndexTreeArray := UINT#204;
                            END_IF;

                            IF statIsLastElement OR statIndexTreeArray + UINT#1 > statTreeLen THEN
                                statIsLastElement := TRUE;
                                statCurrentDepth := 0;
                                statFbState := FB_STATE_CLOSE_STACK_ELEMENT;
                                CONTINUE;
                            ELSIF tree[statIndexTreeArray].types = -1 THEN
                                statCurrentDepth := 0;
                                statIsLastElement := TRUE;
                                statFbState := FB_STATE_CLOSE_STACK_ELEMENT;
                                CONTINUE;
                            END_IF;

                            IF tree[statIndexTreeArray].depth < statCurrentDepth THEN
                                statCurrentDepth := tree[statIndexTreeArray].depth;
                                statFbState := FB_STATE_CLOSE_STACK_ELEMENT;
                                CONTINUE;
                            END_IF;
                            statCurrentDepth := tree[statIndexTreeArray].depth;

                            // The next index would be out of bounds of the tree array
                            // set last element flag and close all stack elements, if there are any
                            IF statIndexTreeArray + UINT#1 > statTreeLen THEN
                                statIsLastElement := TRUE;
                            ELSE
                                // Check if next element is initialized, if not set
                                // last element flag and close all stack elements, if there are any
                                IF tree[statIndexTreeArray + UINT#1].depth = -1
                                    OR tree[statIndexTreeArray + UINT#1].types = -1
                                    OR tree[statIndexTreeArray + UINT#1].key = EMPTY_STRING
                                THEN
                                    statIsLastElement := TRUE;
                                END_IF;

                            END_IF;

                            statFbState := FB_STATE_ELEMENT_TYPE_OPEN;

                            // Overwrite state if the current element is the last element or the next
                            // element has a higher depth.
                            (*
                            IF #statIsLastElement THEN
                                #statFbState := #FB_STATE_CLOSE_STACK_ELEMENT;
                            END_IF;
                            *)

                        //endregion GET NEXT ELEMENT

                    FB_STATE_ELEMENT_TYPE_OPEN: // Check Type and write tree value

                        IF statIndexTreeArray = UINT#45 THEN
                            statIndexTreeArray := UINT#45;
                        END_IF;

                        tempHasNested := FALSE;

                        statInfoToWrite := Concat(string1 := XML_KEY_OPEN,
                                                string2 := tree[statIndexTreeArray].key);

                        tempCntCharsAdded := LStream_WriteOutString(offset := statIndexXmlByteArray, toWrite := statInfoToWrite, xmlByteArray := xmlByteArray);

                        IF tempCntCharsAdded <= -1 THEN
                            statStatus := ERR_XML_OUT_OF_BOUNDS;
                            CONTINUE;
                        END_IF;

                        // Should not loose information as the condition of negative count is a error case
                        // and checked above
                        statIndexXmlByteArray := statIndexXmlByteArray + TO_UINT(tempCntCharsAdded) + UINT#1;

                        tempIterator := statIndexTreeArray;

                        WHILE tempIterator + UINT#1 < statTreeLen DO

                            IF tree[tempIterator + UINT#1].types <> ATTRIBUTE THEN
                                EXIT;
                            END_IF;

                            tempIterator := tempIterator + UINT#1;

                            // Write attribute infos to the string, assuming that they are in combination shorter than the string datatype
                            statInfoToWrite := Concat(string1 := WHITE_SPACE,
                                                string2 := tree[tempIterator].key,
                                                string3 := XML_ATTRIBUTE_OPEN,
                                                string4 := tree[tempIterator].value);
                            /// ADD Temp String because 5 concat is not supported
                            statInfoToWrite := Concat(string1 := statInfoToWrite, string2 := XML_ATTRIBUTE_CLOSE);
                            /*statInfoToWrite := Concat(
                                                              IN1 := WHITE_SPACE,
                                                              IN2 := tree[tempIterator].key,
                                                              IN3 := XML_ATTRIBUTE_OPEN,
                                                              IN4 := tree[tempIterator].value,
                                                              IN5 := XML_ATTRIBUTE_CLOSE);*/

                            tempCntCharsAdded := LStream_WriteOutString(offset := statIndexXmlByteArray, toWrite := statInfoToWrite, xmlByteArray := xmlByteArray);

                            IF tempCntCharsAdded = -1 THEN
                                statStatus := ERR_XML_OUT_OF_BOUNDS;
                                EXIT;
                            END_IF;

                            // Should not loose information as the condition of negative count is a error case
                            // and checked above
                            statIndexXmlByteArray := statIndexXmlByteArray + TO_UINT(tempCntCharsAdded) + UINT#1;

                        END_WHILE;

                        IF statStatus = ERR_XML_OUT_OF_BOUNDS THEN
                            statFbState := FB_STATE_ERROR;
                            CONTINUE;
                        END_IF;

                        IF tempIterator + UINT#1 <= statTreeLen THEN
                            // Has nested elements
                            IF tree[tempIterator + UINT#1].depth > statCurrentDepth THEN
                                IF (TO_DINT(statStackIndex) < STACK_SIZE) THEN
                                    statStackIndex := statStackIndex + TO_INT(INCREMENT_BY_ONE);
                                    statStackIndexOpenElement[statStackIndex] := statIndexTreeArray;
                                    tempHasNested := TRUE;
                                ELSE //Error: Stack out of Bound
                                    statStatus := ERR_STACK_OUT_OF_BOUNDS;
                                    statFbState := FB_STATE_ERROR;
                                    CONTINUE;
                                END_IF;
                            END_IF;
                        ELSE
                            statIsLastElement := TRUE;
                            statFbState := FB_STATE_CLOSE_STACK_ELEMENT;
                            CONTINUE;
                        END_IF;

                        IF tree[statIndexTreeArray].value <> NULL_CONST OR tempHasNested THEN
                            // Write attribute infos to the string, assuming that they are in combination shorter than the string datatype
                            statInfoToWrite := XML_KEY_CLOSE_GREATER;

                            IF tree[statIndexTreeArray].value <> NULL_CONST THEN
                                statInfoToWrite := Concat(string1 := XML_KEY_CLOSE_GREATER, string2 := tree[statIndexTreeArray].value);
                                IF NOT tempHasNested THEN
                                    statInfoToWrite := Concat(string1 := statInfoToWrite,
                                                        string2 := XML_KEY_OPEN,
                                                        string3 := XML_KEY_CLOSE_SLASH);
                                    statInfoToWrite := Concat(string1 := statInfoToWrite,
                                                            string2 := tree[statIndexTreeArray].key,
                                                            string3 := XML_KEY_CLOSE_GREATER);

                                END_IF;
                            END_IF;

                            tempCntCharsAdded := LStream_WriteOutString(offset := statIndexXmlByteArray, toWrite := statInfoToWrite, xmlByteArray := xmlByteArray);

                            IF tempCntCharsAdded = -1 THEN
                                statStatus := ERR_XML_OUT_OF_BOUNDS;
                                statFbState := FB_STATE_ERROR;
                                CONTINUE;
                            END_IF;

                            // Should not loose information as the condition of negative count is a error case
                            // and checked above
                            statIndexXmlByteArray := statIndexXmlByteArray + TO_UINT(tempCntCharsAdded) + UINT#1;

                            // Close element with short form '/>'
                        ELSIF tree[statIndexTreeArray].value = NULL_CONST THEN

                            // This IF considers the situation in which the value of the tree node is 'NULL'
                            IF NOT tempHasNested THEN

                            statInfoToWrite := XML_KEY_CLOSE_GREATER;

                            statInfoToWrite := Concat(string1 := statInfoToWrite,
                                                string2 := XML_KEY_OPEN,
                                                string3 := XML_KEY_CLOSE_SLASH);
                            statInfoToWrite := Concat(string1 := statInfoToWrite,
                                                    string2 := tree[statIndexTreeArray].key,
                                                    string3 := XML_KEY_CLOSE_GREATER);

                            tempCntCharsAdded := LStream_WriteOutString(offset := statIndexXmlByteArray, toWrite := statInfoToWrite, xmlByteArray := xmlByteArray);

                            ELSE

                            // Write attribute infos to the string, assuming that they are in combination shorter than the string datatype
                            statInfoToWrite := Concat(string1 := XML_KEY_CLOSE_SLASH, string2 := XML_KEY_CLOSE_GREATER);
                            tempCntCharsAdded := LStream_WriteOutString(offset := statIndexXmlByteArray, toWrite := statInfoToWrite, xmlByteArray := xmlByteArray);

                            END_IF;

                            IF tempCntCharsAdded = -1 THEN
                                statStatus := ERR_XML_OUT_OF_BOUNDS;
                                statFbState := FB_STATE_ERROR;
                                CONTINUE;
                            END_IF;
                            // Should not loose information as the condition of negative count is a error case
                            // and checked above
                            statIndexXmlByteArray := statIndexXmlByteArray + TO_UINT(tempCntCharsAdded) + UINT#1;

                        END_IF;

                        statIndexTreeArray := tempIterator + UINT#1;
                        statFbState := FB_STATE_NEXT_ELEMENT;
                        CONTINUE;

                    FB_STATE_CLOSE_STACK_ELEMENT: //Close Open Stack Elements
                        //region CLOSE ELEMENT FROM STACK

                            IF statStackIndex < 0 THEN

                                IF statIsLastElement THEN
                                    statFbState := FB_STATE_DONE;
                                ELSE
                                    statFbState := FB_STATE_NEXT_ELEMENT;
                                    statIndexTreeArray := statIndexTreeArray + UINT#1;
                                END_IF;

                                CONTINUE;

                            END_IF;

                            WHILE tree[statStackIndexOpenElement[statStackIndex]].depth >= statCurrentDepth DO

                                // Write attribute infos to the string, assuming that they are in combination shorter than the string datatype
                                statInfoToWrite := Concat(
                                                                  string1 := XML_KEY_OPEN,
                                                                  string2 := XML_KEY_CLOSE_SLASH,
                                                                  string3 := tree[statStackIndexOpenElement[statStackIndex]].key,
                                                                  string4 := XML_KEY_CLOSE_GREATER);

                                tempCntCharsAdded := LStream_WriteOutString(offset := statIndexXmlByteArray, toWrite := statInfoToWrite, xmlByteArray := xmlByteArray);

                                IF tempCntCharsAdded = -1 THEN
                                    statStatus := ERR_XML_OUT_OF_BOUNDS;
                                    EXIT;
                                END_IF;

                                // Should not loose information as the condition of negative count is a error case
                                // and checked above
                                statIndexXmlByteArray := statIndexXmlByteArray + TO_UINT(tempCntCharsAdded) + UINT#1;
                                statWorkingDepth := tree[statStackIndexOpenElement[statStackIndex]].depth;
                                statStackIndexOpenElement[statStackIndex] := UINT#0;
                                statStackIndex := statStackIndex - DECREMENT_BY_ONE;

                                IF statStackIndex < 0 THEN
                                    EXIT;
                                END_IF;

                            END_WHILE;
                            statCurrentDepth := statWorkingDepth;
                            IF statIsLastElement THEN
                                // -> goto stack and close everything until depth = next elements depth
                                statFbState := FB_STATE_DONE;
                            ELSE
                                statFbState := FB_STATE_NEXT_ELEMENT;
                            END_IF;

                        //endregion CLOSE ELEMENT FROM STACK

                    FB_STATE_ERROR:
                        //region STATE ERROR

                            statFbState := FB_STATE_NO_PROCESSING;
                            statError := TRUE;
                            statDone := FALSE;

                        //endregion STATE ERROR;

                    FB_STATE_DONE:
                        //region STATE MACHINE DONE
                            statCount := statIndexXmlByteArray;
                            statDone := FALSE;
                            statStatus := STATUS_EXECUTION_FINISHED;
                            statFbState := FB_STATE_NO_PROCESSING;
                            tempExecute := FALSE;

                        //endregion STATE MACHINE DONE

                    ELSE // Undefined state in state machine reached
                        //REGION UNDEFINED STATE
                            statStatus := ERR_UNDEFINED_STATE;
                        //endregion UNDEFINED STATE

                END_CASE;

                // Call for Timeout timer to update value
                TimeoutTimer();
                //Leave state machine if one of the following condition is true
                //1. state has not changed
                //2. error has occurred
                //3. watchdog timer expired
                //4. execution has finished
                // otherwise stay in state machine
            UNTIL (statFbPreviousState = statFbState OR statStatus.%X15
            OR TimeoutTimer.output OR statStatus = STATUS_EXECUTION_FINISHED)
            END_REPEAT;
        //endregion STATE_MACHINE

    // REGION OUTPUTS
    // Write outputs
    IF (statStatus = STATUS_EXECUTION_FINISHED) AND (statDone = FALSE) THEN // Execution finished without errors
        // REGION EXECUTION FINISHED
            statDone := TRUE;
            statBusy := FALSE;
            statError := FALSE;
            // execution aborted --> set state no processing
            statFbState := FB_STATE_NO_PROCESSING;
        // END_REGION EXECUTION FINISHED

    ELSIF (statStatus.%X15 = TRUE) AND (statError = FALSE) THEN // Error occurred (statStatus is 168000 to 16FFFF)
        // REGION ERROR OCCURRED
            statDone := FALSE;
            statBusy := FALSE;
            statError := TRUE;
            // execution aborted --> set state no processing
            statFbState := FB_STATE_NO_PROCESSING;
        // END_REGION ERROR OCCURRED

    ELSIF (tempExecute = FALSE) AND ((statDone = TRUE) OR (statError = TRUE)) THEN // Reset outputs
        // REGION EXECUTE RESET
            statDone := FALSE;
            statBusy := FALSE;
            statError := FALSE;
            statStatus := STATUS_NO_CALL;
            // Reset application specific outputs
            statCount := UINT#0;
        // END_REGION EXECUTE RESET
    END_IF;

    // REGION WRITE STATIC VALUES TO OUTPUTS
        done := statDone;
        busy := statBusy;
        error := statError;
        status := statStatus;
        // Write application specific static values to outputs
        count := statCount;
    // END_REGION WRITE STATIC VALUES TO OUTPUTS
// END_REGION OUTPUTS

    END_FUNCTION_BLOCK
END_NAMESPACE
